// TIA Portal project "styczeń 2014" (V11)

(* hardware
DEVICE "S7-400 station_1"  S7400.Device
   slot 0: "UR1_0"  UR1  6ES7 400-1TA01-0AA0
   slot 2: "PLC_1"  CPU 416F-3 PN/DP  6ES7 416-3FR05-0AB0  V5.3
      slot 5: "PROFINET interface_1"  PN-IO
         slot 1: "Port_1"  Port
         slot 2: "Port_2"  Port
*)

// ===== PLC "PLC_1"  CPU 416F-3 PN/DP =====

VAR_GLOBAL   // PLC tag table "Default tag table"
   "S1" AT %I0.0 : Bool;
   "IS2" AT %I0.1 : Bool;
   "Tag_3" AT %MW30 : Int;
   "Tag_4" AT %MD2 : DWord;
   "Tag_5" AT %MD3 : DInt;
   "PS" AT %I0.3 : Bool;
   "Tag_7" AT %MW3 : Word;
   "Tag_8" AT %MD30 : Real;
   "Tag_9" AT %MW50 : Int;
   "Tag_10" AT %MW40 : Int;
   "Tag_11" AT %MD50 : Time;
   "Tag_12" AT %MD40 : Time;
   "R" AT %Q0.0 : Bool;
   "Tag_1" AT %M10.0 : Bool;
   "POZYCJA A3" AT %M0.2 : Bool;
   "DOPEŁNIANIE GAZEM" AT %M0.4 : Bool;
   "Tag_2" AT %M5.7 : Bool;
   "Tag_6" AT %M10.7 : Bool;
   "Tag_13" AT %M5.6 : Bool;
   "POZYCJA A2" AT %M0.6 : Bool;
   "CZAS Z KALIBRACJI" AT %MD70 : Time;
   "Tag_14" AT %MW35 : Int;
   "Tag_15" AT %MD20 : DWord;
   "Tag_16" AT %MD55 : Time;
   "Tag_17" AT %MW20 : Int;
   "Tag_18" AT %MD35 : Time;
   "Tag_19" AT %MD80 : DWord;
   "Tag_20" AT %M0.0 : Bool;
   "Tag_21" AT %MW32 : Int;
   "Tag_22" AT %MD11 : DWord;
   "Tag_23" AT %MW48 : Time;
   "Tag_24" AT %MD48 : DWord;
   "BUTLA NIESZCZELNA" AT %M1.2 : Bool;
   "Tag_25" AT %M7.7 : Bool;
   "POZYCJA A1" AT %M1.3 : Bool;
   "Tag_26" AT %M12.2 : Bool;
   "EF" AT %Q0.6 : Bool;
   "BUTLA OK" AT %M1.7 : Bool;
   "Tag_28" AT %M20.1 : Bool;
   "Tag_29" AT %M18.7 : Bool;
   "Tag_30" AT %M6.6 : Bool;
   "BLOKADA NOWEGO CYKLU" AT %M2.3 : Bool;
   "Tag_31" AT %M13.0 : Bool;
   "Tag_32" AT %M13.5 : Bool;
   "FS1" AT %I0.2 : Bool;
   "BLOKADA NAPĘDU" AT %M4.4 : Bool;
   "S2" AT %I0.4 : Bool;
   "ZATRZYMANIE" AT %M1.6 : Bool;
   "Tag_27" AT %Q0.1 : Bool;
   "ED1" AT %Q0.2 : Bool;
   "ED2" AT %Q0.3 : Bool;
   "Tag_33" AT %M6.7 : Bool;
   "Tag_34" AT %MD65 : Time;
END_VAR

ORGANIZATION_BLOCK "Main"   // OB1, LAD
TITLE = "Main Program Sweep (Cycle)"
{ S7_Optimized_Access := 'FALSE' }
VERSION : 0.1
// Wciśnięcie S2 powoduje włączenie stanu zatrzymanie. Wciśnięcie S1 przy niewciśniętym S2 powoduje wyjście ze stanu ZATRZYMANIE
   VAR_TEMP
      OB1_EV_CLASS : Byte;   // Bits 0-3 = 1 (Coming event), Bits 4-7 = 1 (Event class 1)
      OB1_SCAN_1 : Byte;   // 1 (Cold restart scan 1 of OB 1), 3 (Scan 2-n of OB 1)
      OB1_PRIORITY : Byte;   // Priority of OB Execution
      OB1_OB_NUMBR : Byte;   // 1 (Organization block 1, OB1)
      OB1_RESERVED_1 : Byte;   // Reserved for system
      OB1_RESERVED_2 : Byte;   // Reserved for system
      OB1_PREV_CYCLE : Int;   // Cycle time of previous OB1 scan (milliseconds)
      OB1_MIN_CYCLE : Int;   // Minimum cycle time of OB1 (milliseconds)
      OB1_MAX_CYCLE : Int;   // Maximum cycle time of OB1 (milliseconds)
      OB1_DATE_TIME : Date_And_Time;   // Date and time OB1 started
   END_VAR
BEGIN
END_ORGANIZATION_BLOCK